FUNCTION_BLOCK PUBLIC DataParser
VAR_INPUT
	GivenArray : ARRAY[0..5] OF REAL;
END_VAR
VAR_OUTPUT
	OutputArray : ARRAY[0..5] OF REAL;
END_VAR
VAR
	i : INT;
END_VAR

FOR i:= 0 TO 5 BY 1 DO
    OutputArray[i] := ParameterParsingValue(GivenArray[i]);
END_FOR;

END_FUNCTION_BLOCK

(* stored: Version 1.1.0.1, ProductVersion 3.1.4024.0
   POU DataParser: Id {d90a479b-7202-477b-8182-7724e4add93c}, SpecialFunc None *)
